TYPE ST_BaseDescriptor :
STRUCT
	stTexts						: ST_BaseLabel;
	sUnit						: STRING(6);
	rValue						: REAL;
	rMin						: REAL;
	rMax						: REAL;
	rDefaultValue				: REAL;
	
END_STRUCT
END_TYPE

(* stored: Version 1.1.0.1
   DUT ST_BaseDescriptor: Id {6599cd84-8a99-00ca-1312-c67e4a5fcf51} *)
